FUNCTION_BLOCK FB_ComauInterface
VAR_INPUT
	cmnd : DINT;
	control : ST_ComauControl;
END_VAR
VAR_OUTPUT
	feedback : ST_ComauFeedback;
	active : BOOL:= FALSE;
END_VAR
VAR
	// Udp related
	{attribute 'tc_no_symbol'}
	udpClient : FB_UdpClient('', 0, 0, 0, 0, 0, 0);	// Dummy constructor
	rxUdp : ST_RxUdpComau;
	txUdp : ST_TxUdpComau;
	
	pTxHmi : POINTER TO ST_TxHmiComau;
	
	// Actviity monitoring
	frame : DINT := 0;
	frameOld : DINT := 0;
	frameLoss : DINT := 0;
END_VAR

// Check activity
frame := rxUdp.frameCounter;
IF frame <> frameOld THEN
	// Update frame old
	frameOld := frame;
	
	// Reset frameLoss
	frameLoss := 0;
ELSE
	// Count frame losses
	frameLoss := frameLoss + 1;
END_IF

// Set activity status after 1 second given 5ms in ms
IF frameLoss > 200 THEN
	active := FALSE;
ELSE
	active := TRUE;
END_IF

// Update udpClient
udpClient();

// Update Hmi data
UpdateHMI();

// Apply control inputs
txUdp.cmnd := cmnd;
txUdp.udp_key := 32;

txUdp.q1 := LREAL_TO_REAL(control.q[0]);
txUdp.q2 := LREAL_TO_REAL(control.q[1]);
txUdp.q3 := LREAL_TO_REAL(control.q[2]);
txUdp.q4 := 0.0;
txUdp.q5 := 0.0;
txUdp.q6 := 0.0;

txUdp.q1_t := LREAL_TO_REAL(control.q_t[0]);
txUdp.q2_t := LREAL_TO_REAL(control.q_t[1]);
txUdp.q3_t := LREAL_TO_REAL(control.q_t[2]);
txUdp.q4_t := 0.0;
txUdp.q5_t := 0.0;
txUdp.q6_t := 0.0;

txUdp.q1_tt := control.q_tt[0];
txUdp.q2_tt := control.q_tt[1];
txUdp.q3_tt := control.q_tt[2];
txUdp.q4_tt := 0.0;
txUdp.q5_tt := 0.0;
txUdp.q6_tt := 0.0;

// Set feedback data
feedback.q[0] := REAL_TO_LREAL(rxUdp.q1);
feedback.q[1] := REAL_TO_LREAL(rxUdp.q2);
feedback.q[2] := REAL_TO_LREAL(rxUdp.q3);

feedback.q_t[0] := REAL_TO_LREAL(rxUdp.q1_t);
feedback.q_t[1] := REAL_TO_LREAL(rxUdp.q2_t);
feedback.q_t[2] := REAL_TO_LREAL(rxUdp.q3_t);

METHOD FB_exit : BOOL
VAR_INPUT
	bInCopyCode : BOOL; // if TRUE, the exit method is called for exiting an instance that is copied afterwards (online change).
END_VAR
END_METHOD

METHOD FB_init : BOOL
VAR_INPUT
	bInitRetains : BOOL; // if TRUE, the retain variables are initialized (warm start / cold start)
	bInCopyCode : BOOL;  // if TRUE, the instance afterwards gets moved into the copy code (online change)
	
	// Init variables
	_remoteIpAddr : T_Ipv4Addr;
	_remotePort : UINT;
	_localPort : UINT;
	_pTxHmi : POINTER TO ST_TxHmiComau;
END_VAR
pTxHmi := _pTxHmi;

// Initilize udpClient
udpClient.FB_init(
	bInitRetains,
	bInCopyCode,
	_remoteIpAddr,
	_remotePort,
	_localPort,
	SIZEOF(rxUdp),
	ADR(rxUdp),
	SIZEOF(txUdp),
	ADR(txUdp)
);
END_METHOD

METHOD FB_reinit : BOOL
VAR_INPUT
END_VAR
END_METHOD

METHOD UpdateHMI : BOOL
VAR_INPUT
END_VAR
// Update HMI Data
IF active THEN
	pTxHmi^.status := 0;
ELSE
	pTxHmi^.status := -1;
END_IF

pTxHmi^.q[0] := rxUdp.q1;
pTxHmi^.q[1] := rxUdp.q2;
pTxHmi^.q[2] := rxUdp.q3;
pTxHmi^.q[3] := rxUdp.q4;
pTxHmi^.q[4] := rxUdp.q5;
pTxHmi^.q[5] := rxUdp.q6;
END_METHOD

END_FUNCTION_BLOCK

(* stored: Version 1.1.0.1, ProductVersion 3.1.4022.7
   POU FB_ComauInterface: Id {7f6fcfb6-ea5d-4e07-bbf6-5b138a56f61f}, SpecialFunc None
   Method FB_exit: Id {f18839c2-6d63-4a3d-ad66-5f830bcc3ab8}
   Method FB_init: Id {e202aff2-65cb-4030-9293-23617d8046a4}
   Method FB_reinit: Id {09f56272-fe35-4170-800b-7842448d6227}
   Method UpdateHMI: Id {360dfad7-3f26-47be-97c5-29d518768fdd} *)
